FUNCTION_BLOCK XtsHardware
VAR_INPUT
END_VAR
VAR_OUTPUT
END_VAR
VAR
END_VAR

END_FUNCTION_BLOCK

(* stored: Version 1.1.0.1, ProductVersion 3.1.4024.6
   POU XtsHardware: Id {c69630cb-dc63-4ece-b97e-1738681b1044}, SpecialFunc None *)
